# EPICS substitutions: ek9000App/Db/EL1008_mbbiDirect.substitutions
file EL1008.template
{       pattern
        {
                TERMINAL,

        }
        {
        }
}
